{attribute 'Tc2GvlVarNames'}
VAR_GLOBAL CONSTANT
	(* WP_Zustand_Status *)
	E_WP_Zustand_Status_Idle_Sperre					: SINT := 0;
	E_WP_Zustand_Status_Betriebsbereit				: SINT := 1;
	E_WP_Zustand_Status_Nachl						: SINT := 2;
	E_WP_Zustand_Status_Vorl						: SINT := 3;
	E_WP_Zustand_Status_Betrieb						: SINT := 4;
	E_WP_Zustand_Status_Betrieb_Sperre				: SINT := 5;
	E_WP_Zustand_Status_Stoerung					: SINT := 99;

	(* System_WP_Zustand_Status *)
	E_System_WP_Zustand_Status_Idle_Sperre			: SINT := 0;
	E_System_WP_Zustand_Status_Betriebsbereit		: SINT := 1;
	E_System_WP_Zustand_Status_Nachl_Stellventil	: SINT := 2;
	E_System_WP_Zustand_Status_Vorl_Stellventil		: SINT := 3;
	(*E_System_WP_Zustand_Status_Nachl_Pumpe		: SINT := 4;*)
	(*E_System_WP_Zustand_Status_Vorl_Pumpe			: SINT := 5;*)
	E_System_WP_Zustand_Status_Nachl_WP				: SINT := 6;
	E_System_WP_Zustand_Status_Vorl_WP				: SINT := 7;
	E_System_WP_Zustand_Status_Betrieb				: SINT := 8;
	E_System_WP_Zustand_Status_Betrieb_Sperre		: SINT := 9;
	E_System_WP_Zustand_Status_Stoerung				: SINT := 99;
END_VAR

(* stored: Version 1.1.0.1, ProductVersion 3.1.4024.9
   GVL Con_WP: Id {9cfaec1e-4a9e-4898-bf0b-606a5c5d94d0} *)
